Fanuc KAREL source: ko00072.KL

-- PROVISIONAL review KL for V1013-1; original PC SHA256 276a4a06e3bf87812c0002a70ad78b5499f539aefe0727871522e0fd4b806e52
-- Incomplete behavior may be omitted. Consult companion uncertainty JSON. Do not deploy.
PROGRAM KO00072
%NOLOCKGROUP
BEGIN
  -- UNRESOLVED_PC offsets 5-12; opcodes 9D,23
  -- UNRESOLVED_PC offsets 17-66; opcodes 27,22,1C,27,49,7E,AD,22,31,7E,4A
  -- UNRESOLVED_PC offsets 71-75; opcodes 7F
END KO00072
